# B&R Automation Studio project Sim_Eksamen_Test1
Automation Studio 4.7.2.98

## Logical view

### Global.typ - Global data types
```iecst
(*Denne Type er de 2 stadier som vores robot arm kan befinde sig i.*)

TYPE
	RobotArm : 	STRUCT
		Getting : BOOL;
		Delivering : BOOL;
	END_STRUCT;
END_TYPE
```

### Program Logical/Sorter (IEC)

#### Variables.var
```iecst
VAR
	doSorterPick : BOOL;
	diRightPos : BOOL;
	diPos2OutOfPlace : BOOL;
	diPos1OutOfPlace : BOOL;
	diPos1OutOfPlaceWeight : INT;
	diPos2OutOfPlaceWeight : INT;
	diWeightScale : WORD;
	R_TRIG_RightPos : R_TRIG;
	R_TRIG_PickInitiated : R_TRIG;
	TON_OffTimer : TON;
	TON_DelayTimer : TON;
	sorterRobot : RobotArm;
	bigBoxDetected : BOOL;
END_VAR
```

#### Main.st
```iecst
PROGRAM _INIT
	// Timer initialization
	TON_DelayTimer.PT := T#1s;
END_PROGRAM

PROGRAM _CYCLIC
	R_TRIG_RightPos.CLK := bigBoxDetected;
	R_TRIG_PickInitiated.CLK := sorterRobot.Delivering;
	// Detecting bigBox
	IF diWeightScale > 300 THEN
		bigBoxDetected := TRUE;
	ELSE
		bigBoxDetected := FALSE;
	END_IF;

	IF diGoBtn THEN

		// Weight gets activated.
		IF R_TRIG_RightPos.Q  THEN
			// If it's notv right, then we pick
			TON_DelayTimer.IN := TRUE;
		END_IF;

		// Delay timer for activating Sorter
		IF TON_DelayTimer.Q THEN
			TON_DelayTimer.IN := FALSE;
			doSorterPick := TRUE;
		END_IF;

		// Delay timer for switching input off. (Might be error if Blocks are too close to one another)
		IF R_TRIG_PickInitiated.Q THEN
			doSorterPick := FALSE;
		END_IF;

	ELSE
		// Reset all.
		TON_DelayTimer.IN := FALSE;
		doSorterPick := FALSE;

	END_IF;

	// Functionblock Calls
	TON_DelayTimer();
	R_TRIG_PickInitiated();
	R_TRIG_RightPos();
END_PROGRAM

PROGRAM _EXIT
	(* Insert code here *)

END_PROGRAM
```

### Program Logical/Stacker (IEC)

#### Variables.var
```iecst
VAR
	doStackerPick : BOOL;
	diStackDone : BOOL;
	R_TRIG_diGoBtn : R_TRIG;
	pickerRobotRight : RobotArm;
	pickerRobotLeft : RobotArm;
	R_TRIG_StackerCount : R_TRIG;
	R_TRIG_StackDone : R_TRIG;
	doConvSideStart : BOOL;
	diPlateBoxBlocked : BOOL;
	F_TRIG_StackDone : F_TRIG;
	F_TRIG_BoxBlocked : F_TRIG;
	doStackerInputBelt : BOOL;
	diStackerInputSensor : BOOL;
	stackCount : USINT;
	doResetStackers : BOOL;
END_VAR
```

#### Main.st
```iecst
PROGRAM _INIT
		(* Insert code here *)

END_PROGRAM

PROGRAM _CYCLIC
	R_TRIG_StackDone.CLK := diStackDone;
	R_TRIG_diGoBtn.CLK := diGoBtn;
	F_TRIG_BoxBlocked.CLK := diPlateBoxBlocked;
	R_TRIG_StackerCount.CLK := diStackerInputSensor;
	F_TRIG_StackDone.CLK := diStackDone;

	IF diGoBtn THEN
		// Stop belt when box is exactly in place.
		doStackerInputBelt := NOT diStackerInputSensor;

		// Increase count on rising edge.
		IF R_TRIG_StackerCount.Q THEN
			stackCount := stackCount +1;
		END_IF;

		// Initiate plate serving in start of program.
		IF R_TRIG_diGoBtn.Q THEN
			doConvSideStart := TRUE;
		END_IF;

		// Move output belt when the stack is stacked,
		IF R_TRIG_StackDone.Q THEN
			doConvSideStart := TRUE;
		END_IF;
		// and stop it again.
		IF F_TRIG_BoxBlocked.Q THEN
			doConvSideStart := FALSE;
			// Reset count according to wether a block is ready for pickup or not.
			IF diStackerInputSensor THEN
				stackCount := 1;
			ELSE
				stackCount := 0;
			END_IF;

			// Reset for stackers
			IF diStackDone THEN
				doResetStackers := TRUE;
			END_IF;
		END_IF;

		// Activate stackers
		doStackerPick := diStackerInputSensor AND
						 NOT (stackCount > 8) AND
						 NOT doConvSideStart AND
						 NOT diStackDone;

		// Reset stacker Reset
		IF F_TRIG_StackDone.Q THEN
			doResetStackers := FALSE;
		END_IF;
	ELSE
		// Reset all.
		doStackerPick := FALSE;
		doConvSideStart := FALSE;
		doStackerInputBelt := FALSE;
		stackCount := 0;
	END_IF;

	// Functionblock Calls
	R_TRIG_StackDone();
	R_TRIG_diGoBtn();
	F_TRIG_BoxBlocked();
	R_TRIG_StackerCount();
	F_TRIG_StackDone();
END_PROGRAM

PROGRAM _EXIT
	(* Insert code here *)

END_PROGRAM
```

Listed in the project but not available here: Logical/Global.var, Logical/Libraries, Logical/Feed_Conv
